{attribute 'qualified_only'}
VAR_GLOBAL
	location : STRING;
	groupId : UDINT;
	axisId1 : UDINT;
	axisId2 : UDINT;
	axisId3 : UDINT;
	timeout : TIME;
	busy : BOOL;
	error : BOOL;
	errorId : UDINT;
	executeCounter : ULINT;
END_VAR

(* stored: Version 1.1.0.1, ProductVersion 3.1.4024.12
   GVL Debug: Id {270af060-0cde-4789-9fa4-1206361762df} *)
